// TIA Portal V20 export
ORGANIZATION_BLOCK "Main"   // OB1001, LAD, ProgramCycle
TITLE = "Main Program Sweep (Cycle)"
// This block calls the FB CallUnit which includes all further functionality of the unit.
// It reads the general global status and the safety status from the respective safety zone.
// It writes the unit status back to the DB Global.Data and the acknowledge information to the respetive safety zone.
// OB Main is a program cycle OB and is called depending on its number. For details, refer to the Automation Framework documentation.
// stored: AutoNumber false, IsIECCheckEnabled true, Namespace Unit1, SetENOAutomatically true
   VAR_INPUT
      Initial_Call : Bool;   // Initial call of this OB
      Remanence : Bool;   // =True, if remanent data are available
   END_VAR
   VAR_TEMP
      tempIndex : Int;   // Index of Unit in the array
   END_VAR
   VAR CONSTANT
      "Temporary bit" : Bool := true;
   END_VAR
BEGIN

REGION Network 1: Call Unit
   // Assign the number of the unit to a temp for correct array index access.
   // Number is defined in PLC tags of Software Unit Global.
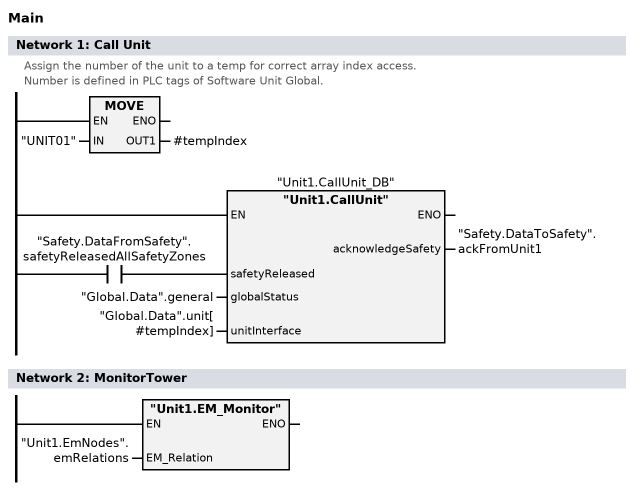
   RUNG wire#powerrail
      Move(in := "UNIT01", out1 => #tempIndex)
   END_RUNG
   RUNG wire#powerrail
      "Unit1.CallUnit_DB"(safetyReleased := wire#w1, globalStatus := "Global.Data".general, unitInterface := "Global.Data".unit[#tempIndex], acknowledgeSafety => "Safety.DataToSafety".ackFromUnit1)
   END_RUNG
   RUNG wire#powerrail
      Contact( "Safety.DataFromSafety".safetyReleasedAllSafetyZones )
   END_RUNG wire#w1
   // the same network as SCL:
   #tempIndex := "UNIT01";
   "Unit1.CallUnit_DB"(safetyReleased := "Safety.DataFromSafety".safetyReleasedAllSafetyZones,   // "Unit1.CallUnit"
                       globalStatus := "Global.Data".general,
                       unitInterface := "Global.Data".unit[#tempIndex],
                       acknowledgeSafety => "Safety.DataToSafety".ackFromUnit1);
END_REGION

REGION Network 2: MonitorTower
   RUNG wire#powerrail
      "Unit1.EM_Monitor"(EM_Relation := "Unit1.EmNodes".emRelations)
   END_RUNG
   // the same network as SCL:
   "Unit1.EM_Monitor"(EM_Relation := "Unit1.EmNodes".emRelations);
END_REGION

REGION Network 3 (SCL): Temp Simulation

   (* IF EmNodes.unitStatus.simulationActive THEN
       IF EmNodes.BA030.StackToInspection.InterfaceData."Bool"[17] THEN
           EmData.partData.transferPnPLeft.Common.LastLegNumber := 'A';
           EmData.partData.sideTape.Common.LastLegNumber := 'A';
       ELSIF EmNodes.BA040.StackToInspection.InterfaceData."Bool"[17] THEN
           EmData.partData.transferPnPLeft.Common.LastLegNumber := 'B';
           EmData.partData.sideTape.Common.LastLegNumber := 'B';
       END_IF;
   END_IF; *)



   IF "JB_Temp".Local_mode THEN
       "Global.Data".unit[0].enableControlInterfaces.hmi := FALSE;
       "Global.Data".unit[0].enableControlInterfaces.local := true;

   END_IF;

   IF "JB_Temp".Test_bypass_Bit AND "JB_Temp".Simulation_initializing THEN

       "Global.Data".unit[0].enableControlInterfaces.hmi :=
       "Global.Data".unit[0].enableControlInterfaces.hmi := true;

       "Global.Data".unit[0].enableControlInterfaces."local" :=
       "Global.Data".unit[0].enableControlInterfaces.remote := false;

       "JB_Temp".Test_Homing[0] :=
       "JB_Temp".Test_Homing[1] :=
       "JB_Temp".Test_Homing[2] :=
       "JB_Temp".Test_Homing[3] :=
       "JB_Temp".Test_Homing[4] :=
       "JB_Temp".Test_Homing[5] :=
       "JB_Temp".Test_Homing[6] :=
       "JB_Temp".Test_Homing[7] :=
       "JB_Temp".Test_Homing[8] :=
       "JB_Temp".Test_Homing[9] :=
       "JB_Temp".Test_Homing[10] :=
       "JB_Temp".Test_Homing[11] :=
       "JB_Temp".Test_Homing[12] :=
       "JB_Temp".Test_Homing[13] := true;

   END_IF;

   (*
   IF _.JB_Temp.Step_by_Step AND EmNodes.unitStatus.simulationActive THEN

       _.JB_Temp.Test_sig_2[1, 2] :=
       _.JB_Temp.Test_sig_2[1, 3] :=
       _.JB_Temp.Test_sig_3[3, 2] :=
       _.JB_Temp.Test_sig_2[1, 4] :=
       _.JB_Temp.Test_sig_3[3, 3] :=
       _.JB_Temp.Test_sig_3[2, 3] :=
       _.JB_Temp.Test_sig_3[3, 4] :=
       _.JB_Temp.Test_sig_3[2, 4] :=
       _.JB_Temp.Test_sig_2[2, 2] :=
       _.JB_Temp.Test_sig_3[3, 5] :=
       _.JB_Temp.Test_sig_3[3, 2] :=
       _.JB_Temp.Test_sig_2[2, 3] :=
       _.JB_Temp.Test_sig_4[3, 2] :=
       _.JB_Temp.Test_sig_4[3, 3] :=
       _.JB_Temp.Test_sig_4[2, 4] :=
       _.JB_Temp.Test_sig_4[3, 4,0] :=
       _.JB_Temp.Test_sig_4[2, 5,0] :=
       _.JB_Temp.Test_sig_4[3, 5,0] :=
       _.JB_Temp.Test_sig_4[2, 6,0] :=
       _.JB_Temp.Test_sig_4[3, 6,0] :=
       _.JB_Temp.Test_sig_4[2, 7,0] :=
       _.JB_Temp.Test_sig_4[3, 7,0] :=
       _.JB_Temp.Test_sig_5[1, 2,0] :=
       _.JB_Temp.Test_sig_6[2,0] :=
       _.JB_Temp.Test_sig_5[1, 3,0] :=
       _.JB_Temp.Test_sig_5[1, 4,0] :=
       _.JB_Temp.Test_sig_5[1, 5,0] :=
       _.JB_Temp.Test_sig_7[2,0] :=
       _.JB_Temp.Test_sig_5[1, 6,0] :=
       _.JB_Temp.Test_sig_5[1, 7,0] :=
       _.JB_Temp.Test_sig_8[1, 2] :=
       _.JB_Temp.Test_sig_5[1, 9,0] :=
       _.JB_Temp.Test_sig_8[1, 4] :=
       _.JB_Temp.Test_sig_5[2, 2,0] :=
       _.JB_Temp.Test_sig_9[1, 2] :=
       _.JB_Temp.Test_sig_5[2, 3,0] :=
       _.JB_Temp.Test_sig_9[1, 4] :=
       _.JB_Temp.Test_sig_5[2, 4,0] :=
       _.JB_Temp.Test_sig_10[2] :=
       _.JB_Temp.Test_sig_5[2, 5,0] :=
       _.JB_Temp.Test_sig_10[4] :=
       _.JB_Temp.Test_sig_5[2, 6,0] :=
       _.JB_Temp.Test_sig_11[2] :=
       _.JB_Temp.Test_sig_5[2, 9,0] :=
       _.JB_Temp.Test_sig_11[4] :=
       _.JB_Temp.Test_sig_13[2,0] := true;

       _.JB_Temp.Step_by_Step := false;
   END_IF;
   *)
END_REGION
END_ORGANIZATION_BLOCK
